(* IEC 61131-3 sources: plc_on_fpga_riscv_hybrid/RV_FPGA_PLC_IDE_Projects/Two_Branches_One_Output, 1 file *)

(* ---- Two_Branches_One_Output.il ---- *)
VAR
END_VAR

PROGRAM Two_Branches_One_Output
    R1 :
        LD     %SW.1
        AND    %SW.2
        OR     (
        LD     %SW.3
        AND    %SW.4
        )
        ST     %LEDG.0
END_PROGRAM
